(* Schneider Machine Expert - Basic project Step13_TrafficMode11_Auto_Ok, file version 1.8.0.0 *)
(* ProjectInformations: Name=New project *)

HARDWARE
  Cpu 0: TM221CE16R
  EthernetConfiguration: NetworkName=M221, IpAllocationMode=FixedAddress, IpAddress=192.168.1.58, SubnetMask=255.255.255.0
  SerialLineConfiguration: Baud=Baud9600, Parity=ParityNone, DataBits=DataBits8, StopBits=StopBits1, PhysicalMedium=PhysicalMediumRs485, TransmissionMode=TransmissionModeModbusRtu, SlaveId=1, Addressing=SlaveAddressing
  MastTask: UsePeriodScanMode=false, PeriodScan=100
  FastTask: Period=255
  CpuBehavior: StartingMode=StartAsPreviousState, AutoSaveRamOnEeprom=true, WatchdogPeriod=250

SYMBOLS  (address, symbol, comment, settings)
  %M0       RMODE_SW
  %M1       RMODE_MSB
  %M2       RMODE_LSB
  %M3       RMANUAL_SW
  %M20      RLED_RED
  %M21      RLED_YLW
  %M22      RLED_GRN
  %TM0      MAN_TIMER  [Preset=1, Base=OneSecond]
  %TM1      BLINK_ON  [Preset=1, Base=OneSecond]
  %TM2      BLINK_OFF  [Preset=1, Base=OneSecond]
  %TM3      DLY_GRN  [Preset=2, Base=OneSecond]
  %TM4      DLY_YLW  [Preset=1, Base=OneSecond]
  %TM5      DLY_RED  [Preset=3, Base=OneSecond]
  %I0.0     SW_GRN  "Sw_GRN"
  %I0.1     SW_BLK
  %Q0.0     LED_RED  "LED_RED"
  %Q0.1     LED_YLW  "LED_YLW"
  %Q0.2     LED_GRN  "LED_GRN"
  %Q0.5     LED_MSB
  %Q0.6     LED_LSB

POU ModeSelect
  (* SectionNumber=1 *)

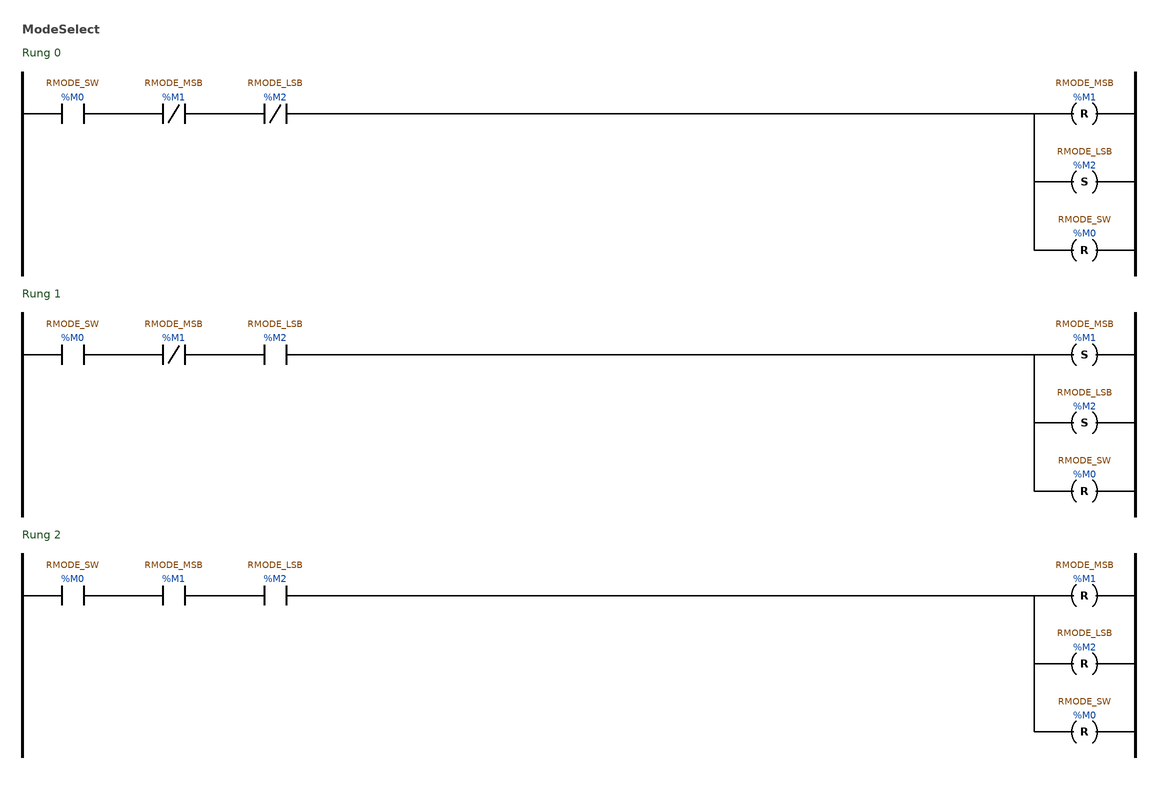

// Rung 0
  LD %M0                  (* RMODE_SW *)
  ANDN %M1                (* RMODE_MSB *)
  ANDN %M2                (* RMODE_LSB *)
  R %M1                   (* RMODE_MSB *)
  S %M2                   (* RMODE_LSB *)
  R %M0                   (* RMODE_SW *)
  // as ST:
  //   _t1 := RMODE_SW AND NOT RMODE_MSB AND NOT RMODE_LSB;
  //   IF _t1 THEN RMODE_MSB := FALSE; END_IF;
  //   IF _t1 THEN RMODE_LSB := TRUE; END_IF;
  //   IF _t1 THEN RMODE_SW := FALSE; END_IF;

// Rung 1
  LD %M0                  (* RMODE_SW *)
  ANDN %M1                (* RMODE_MSB *)
  AND %M2                 (* RMODE_LSB *)
  S %M1                   (* RMODE_MSB *)
  S %M2                   (* RMODE_LSB *)
  R %M0                   (* RMODE_SW *)
  // as ST:
  //   _t1 := RMODE_SW AND NOT RMODE_MSB AND RMODE_LSB;
  //   IF _t1 THEN RMODE_MSB := TRUE; END_IF;
  //   IF _t1 THEN RMODE_LSB := TRUE; END_IF;
  //   IF _t1 THEN RMODE_SW := FALSE; END_IF;

// Rung 2
  LD %M0                  (* RMODE_SW *)
  AND %M1                 (* RMODE_MSB *)
  AND %M2                 (* RMODE_LSB *)
  R %M1                   (* RMODE_MSB *)
  R %M2                   (* RMODE_LSB *)
  R %M0                   (* RMODE_SW *)
  // as ST:
  //   _t1 := RMODE_SW AND RMODE_MSB AND RMODE_LSB;
  //   IF _t1 THEN RMODE_MSB := FALSE; END_IF;
  //   IF _t1 THEN RMODE_LSB := FALSE; END_IF;
  //   IF _t1 THEN RMODE_SW := FALSE; END_IF;

POU Mode11Auto
  (* SectionNumber=2 *)

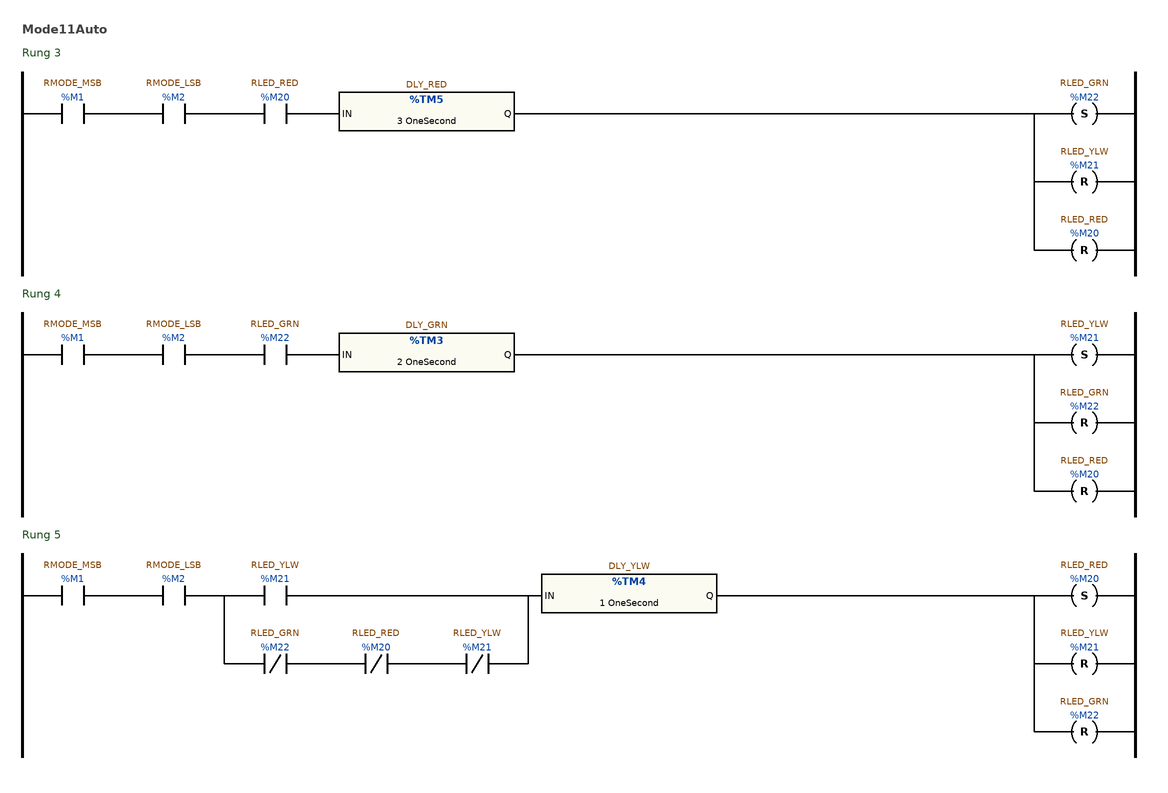

// Rung 3
  BLK %TM5                (* DLY_RED *)
  LD %M1                  (* RMODE_MSB *)
  AND %M2                 (* RMODE_LSB *)
  AND %M20                (* RLED_RED *)
  IN
  OUT_BLK
  LD Q
  S %M22                  (* RLED_GRN *)
  R %M21                  (* RLED_YLW *)
  R %M20                  (* RLED_RED *)
  END_BLK
  // as ST:
  //   DLY_RED(IN := RMODE_MSB AND RMODE_LSB AND RLED_RED);
  //   IF DLY_RED.Q THEN RLED_GRN := TRUE; END_IF;
  //   IF DLY_RED.Q THEN RLED_YLW := FALSE; END_IF;
  //   IF DLY_RED.Q THEN RLED_RED := FALSE; END_IF;

// Rung 4
  BLK %TM3                (* DLY_GRN *)
  LD %M1                  (* RMODE_MSB *)
  AND %M2                 (* RMODE_LSB *)
  AND %M22                (* RLED_GRN *)
  IN
  OUT_BLK
  LD Q
  S %M21                  (* RLED_YLW *)
  R %M22                  (* RLED_GRN *)
  R %M20                  (* RLED_RED *)
  END_BLK
  // as ST:
  //   DLY_GRN(IN := RMODE_MSB AND RMODE_LSB AND RLED_GRN);
  //   IF DLY_GRN.Q THEN RLED_YLW := TRUE; END_IF;
  //   IF DLY_GRN.Q THEN RLED_GRN := FALSE; END_IF;
  //   IF DLY_GRN.Q THEN RLED_RED := FALSE; END_IF;

// Rung 5
  BLK %TM4                (* DLY_YLW *)
  LD %M1                  (* RMODE_MSB *)
  AND %M2                 (* RMODE_LSB *)
  AND( %M21               (* RLED_YLW *)
  OR(N %M22               (* RLED_GRN *)
  ANDN %M20               (* RLED_RED *)
  ANDN %M21               (* RLED_YLW *)
  )
  )
  IN
  OUT_BLK
  LD Q
  S %M20                  (* RLED_RED *)
  R %M21                  (* RLED_YLW *)
  R %M22                  (* RLED_GRN *)
  END_BLK
  // as ST:
  //   DLY_YLW(IN := RMODE_MSB AND RMODE_LSB AND (RLED_YLW OR NOT RLED_GRN AND NOT RLED_RED AND NOT RLED_YLW));
  //   IF DLY_YLW.Q THEN RLED_RED := TRUE; END_IF;
  //   IF DLY_YLW.Q THEN RLED_YLW := FALSE; END_IF;
  //   IF DLY_YLW.Q THEN RLED_GRN := FALSE; END_IF;

POU Mode10Ylw
  (* SectionNumber=3 *)

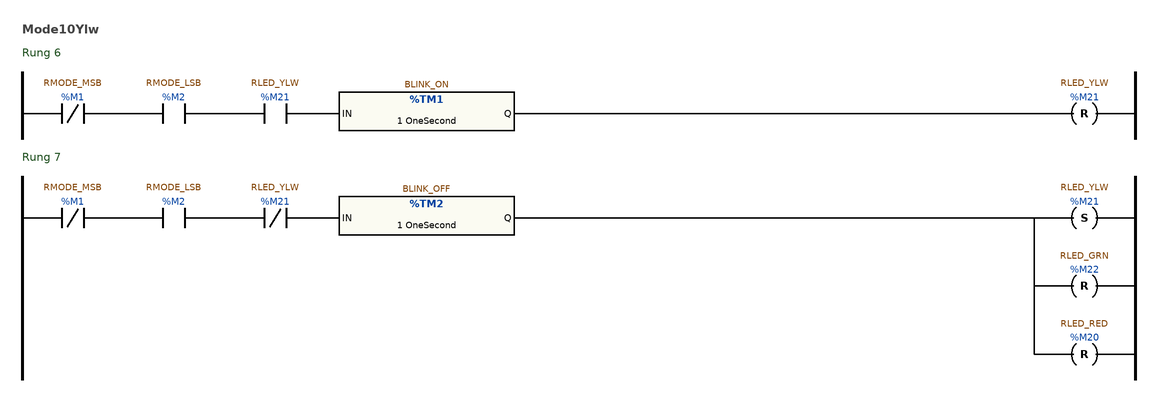

// Rung 6
  BLK %TM1                (* BLINK_ON *)
  LDN %M1                 (* RMODE_MSB *)
  AND %M2                 (* RMODE_LSB *)
  AND %M21                (* RLED_YLW *)
  IN
  OUT_BLK
  LD Q
  R %M21                  (* RLED_YLW *)
  END_BLK
  // as ST:
  //   BLINK_ON(IN := NOT RMODE_MSB AND RMODE_LSB AND RLED_YLW);
  //   IF BLINK_ON.Q THEN RLED_YLW := FALSE; END_IF;

// Rung 7
  BLK %TM2                (* BLINK_OFF *)
  LDN %M1                 (* RMODE_MSB *)
  AND %M2                 (* RMODE_LSB *)
  ANDN %M21               (* RLED_YLW *)
  IN
  OUT_BLK
  LD Q
  S %M21                  (* RLED_YLW *)
  R %M22                  (* RLED_GRN *)
  R %M20                  (* RLED_RED *)
  END_BLK
  // as ST:
  //   BLINK_OFF(IN := NOT RMODE_MSB AND RMODE_LSB AND NOT RLED_YLW);
  //   IF BLINK_OFF.Q THEN RLED_YLW := TRUE; END_IF;
  //   IF BLINK_OFF.Q THEN RLED_GRN := FALSE; END_IF;
  //   IF BLINK_OFF.Q THEN RLED_RED := FALSE; END_IF;

POU Mode00Manual
  (* SectionNumber=4 *)

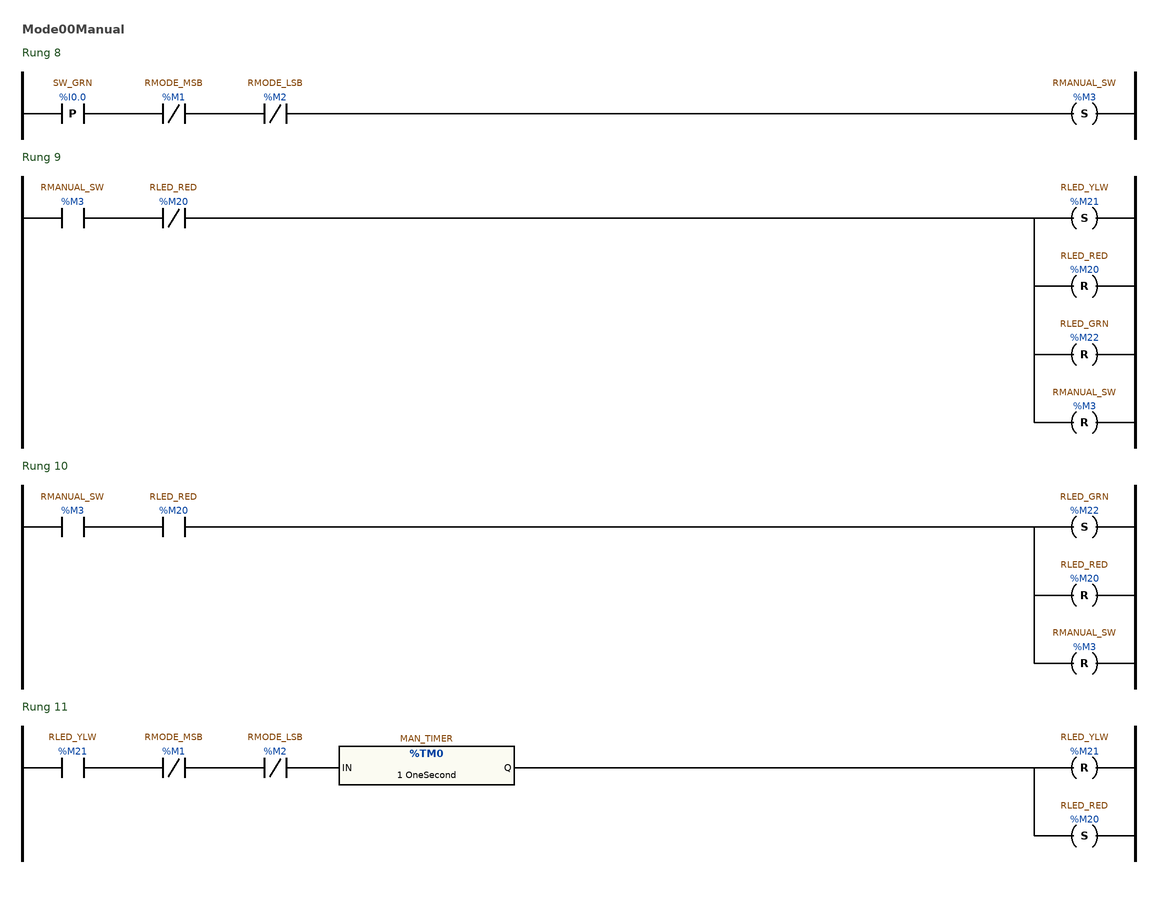

// Rung 8
  LDR %I0.0               (* SW_GRN *)
  ANDN %M1                (* RMODE_MSB *)
  ANDN %M2                (* RMODE_LSB *)
  S %M3                   (* RMANUAL_SW *)
  // as ST:
  //   IF RISING(SW_GRN) AND NOT RMODE_MSB AND NOT RMODE_LSB THEN RMANUAL_SW := TRUE; END_IF;

// Rung 9
  LD %M3                  (* RMANUAL_SW *)
  ANDN %M20               (* RLED_RED *)
  S %M21                  (* RLED_YLW *)
  R %M20                  (* RLED_RED *)
  R %M22                  (* RLED_GRN *)
  R %M3                   (* RMANUAL_SW *)
  // as ST:
  //   IF RMANUAL_SW AND NOT RLED_RED THEN RLED_YLW := TRUE; END_IF;
  //   _t1 := RMANUAL_SW AND NOT RLED_RED;
  //   IF _t1 THEN RLED_RED := FALSE; END_IF;
  //   IF _t1 THEN RLED_GRN := FALSE; END_IF;
  //   IF _t1 THEN RMANUAL_SW := FALSE; END_IF;

// Rung 10
  LD %M3                  (* RMANUAL_SW *)
  AND %M20                (* RLED_RED *)
  S %M22                  (* RLED_GRN *)
  R %M20                  (* RLED_RED *)
  R %M3                   (* RMANUAL_SW *)
  // as ST:
  //   IF RMANUAL_SW AND RLED_RED THEN RLED_GRN := TRUE; END_IF;
  //   _t1 := RMANUAL_SW AND RLED_RED;
  //   IF _t1 THEN RLED_RED := FALSE; END_IF;
  //   IF _t1 THEN RMANUAL_SW := FALSE; END_IF;

// Rung 11
  BLK %TM0                (* MAN_TIMER *)
  LD %M21                 (* RLED_YLW *)
  ANDN %M1                (* RMODE_MSB *)
  ANDN %M2                (* RMODE_LSB *)
  IN
  OUT_BLK
  LD Q
  R %M21                  (* RLED_YLW *)
  S %M20                  (* RLED_RED *)
  END_BLK
  // as ST:
  //   MAN_TIMER(IN := RLED_YLW AND NOT RMODE_MSB AND NOT RMODE_LSB);
  //   IF MAN_TIMER.Q THEN RLED_YLW := FALSE; END_IF;
  //   IF MAN_TIMER.Q THEN RLED_RED := TRUE; END_IF;

POU InputOutput
  (* SectionNumber=5 *)

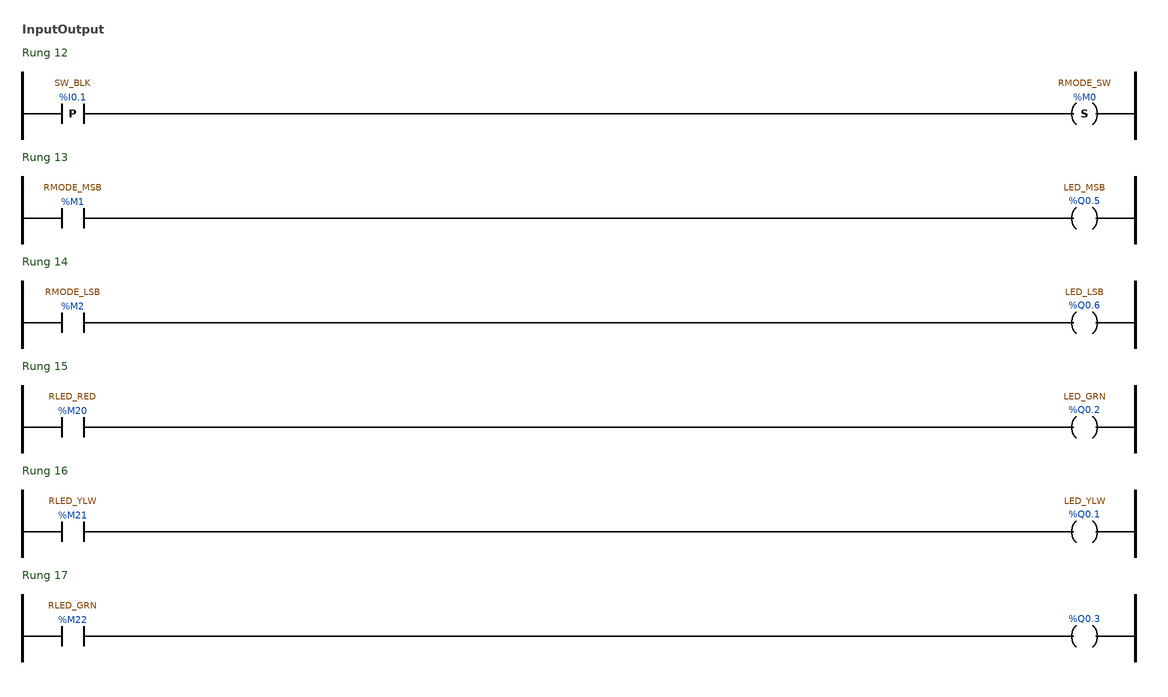

// Rung 12
  LDR %I0.1               (* SW_BLK *)
  S %M0                   (* RMODE_SW *)
  // as ST:
  //   IF RISING(SW_BLK) THEN RMODE_SW := TRUE; END_IF;

// Rung 13
  LD %M1                  (* RMODE_MSB *)
  ST %Q0.5                (* LED_MSB *)
  // as ST:
  //   LED_MSB := RMODE_MSB;

// Rung 14
  LD %M2                  (* RMODE_LSB *)
  ST %Q0.6                (* LED_LSB *)
  // as ST:
  //   LED_LSB := RMODE_LSB;

// Rung 15
  LD %M20                 (* RLED_RED *)
  ST %Q0.2                (* LED_GRN *)
  // as ST:
  //   LED_GRN := RLED_RED;

// Rung 16
  LD %M21                 (* RLED_YLW *)
  ST %Q0.1                (* LED_YLW *)
  // as ST:
  //   LED_YLW := RLED_YLW;

// Rung 17
  LD %M22                 (* RLED_GRN *)
  ST %Q0.3
  // as ST:
  //   %Q0.3 := RLED_GRN;
